TYPE "MachineInterface"
VERSION : 0.1
// Block: MachineInterface
   STRUCT
      AutReady : Bool;
      Aborting : Bool;
      AckStopInPhase : Bool;
      AckStopProgrammed : Bool;
      MotionsStandStill : Bool;
      AlarmsPresence : Bool;
      WarningPresence : Bool;
   END_STRUCT;

END_TYPE
